FUNCTION_BLOCK IN_PAINT (* A drop-down list to select a key to a java.awt.Paint from the GraphComponent hashtable *)
  (* Standard: 61499-1; ApplicationDomain: GUI; Function: java.awt.Paint key input *)
  (* Version 0.0, 2006-12-06, JHC, Holobloc Inc, Derived from IN_COLOR. *)
  (* Compiler header: package fb.rt.gui; import java.awt.*; import java.awt.event.*; *)
  (* Compiler Java IBM VisualAge 3.0 *)
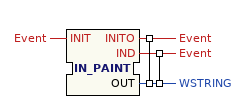
  EVENT_INPUT
    INIT; (* Initialization *)
  END_EVENT
  EVENT_OUTPUT
    INITO WITH OUT; (* Initialization Confirm *)
    IND WITH OUT; (* User Entered Data or REQ was processed *)
  END_EVENT
  VAR_OUTPUT
    OUT : WSTRING;
  END_VAR
END_FUNCTION_BLOCK
